TYPE ST_ShuttleForkData :
STRUCT	
	ForkStatus				: ST_ForkState;
	ForkRequest				: ST_ForkRequest;	
END_STRUCT
END_TYPE

(* stored: Version 1.1.0.1, ProductVersion 3.1.4024.9
   DUT ST_ShuttleForkData: Id {9320fc85-d4a3-499e-bf5a-ce837000e0db} *)
